// TIA Portal project "licznik-silownik" (V11)

(* hardware
DEVICE "S7-400 station_1"  S7400.Device
   slot 0: "UR1_0"  UR1  6ES7 400-1TA01-0AA0
   slot 2: "PLC_1"  CPU 416F-3 PN/DP  6ES7 416-3FR05-0AB0  V5.3
      slot 5: "PROFINET interface_1"  PN-IO
         slot 1: "Port_1"  Port
         slot 2: "Port_2"  Port
*)

// ===== PLC "PLC_1"  CPU 416F-3 PN/DP =====

VAR_GLOBAL   // PLC tag table "Default tag table"
   "Tag_1" AT %M0.0 : Bool;
   "Tag_2" AT %I0.0 : Bool;
   "Tag_3" AT %I0.1 : Bool;
   "Tag_4" AT %M1.0 : Bool;
   "Tag_5" AT %T1 : Timer;
   "Tag_6" AT %Q0.0 : Bool;
   "Tag_7" AT %M0.1 : Bool;
   "Tag_8" AT %M0.2 : Bool;
   "Tag_9" AT %I0.2 : Bool;
END_VAR

ORGANIZATION_BLOCK "Main"   // OB1, LAD
TITLE = "Main Program Sweep (Cycle)"
{ S7_Optimized_Access := 'FALSE' }
VERSION : 0.1
   VAR_TEMP
      OB1_EV_CLASS : Byte;   // Bits 0-3 = 1 (Coming event), Bits 4-7 = 1 (Event class 1)
      OB1_SCAN_1 : Byte;   // 1 (Cold restart scan 1 of OB 1), 3 (Scan 2-n of OB 1)
      OB1_PRIORITY : Byte;   // Priority of OB Execution
      OB1_OB_NUMBR : Byte;   // 1 (Organization block 1, OB1)
      OB1_RESERVED_1 : Byte;   // Reserved for system
      OB1_RESERVED_2 : Byte;   // Reserved for system
      OB1_PREV_CYCLE : Int;   // Cycle time of previous OB1 scan (milliseconds)
      OB1_MIN_CYCLE : Int;   // Minimum cycle time of OB1 (milliseconds)
      OB1_MAX_CYCLE : Int;   // Maximum cycle time of OB1 (milliseconds)
      OB1_DATE_TIME : Date_And_Time;   // Date and time OB1 started
   END_VAR
   VAR_TEMP   // added for the SCL form of the ladder/FBD networks
      _w1 : Bool;
      _s5time1 : S5Time;
   END_VAR
BEGIN

REGION Network 1
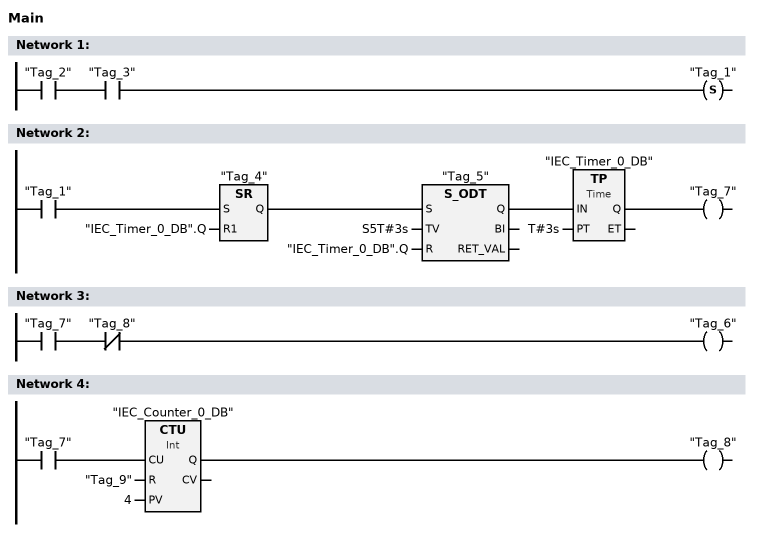
   RUNG wire#powerrail
      Contact( "Tag_2" )
      Contact( "Tag_3" )
      S_Coil( "Tag_1" )
   END_RUNG
   // the same network as SCL:
   IF "Tag_2" AND "Tag_3" THEN "Tag_1" := TRUE; END_IF;
END_REGION

REGION Network 2
   IF "Tag_1" THEN
       "Tag_4" := TRUE;   // SR flip-flop
   END_IF;
   IF "IEC_Timer_0_DB".Q THEN "Tag_4" := FALSE; END_IF;
   #_s5time1 := S_ODT(T_NO := "Tag_5", S := "Tag_4", TV := S5T#3s, R := "IEC_Timer_0_DB".Q, Q => #_w1);
   "IEC_Timer_0_DB".TP(IN := #_w1, PT := T#3s);
   "Tag_7" := "IEC_Timer_0_DB".Q;
END_REGION

REGION Network 3
   RUNG wire#powerrail
      Contact( "Tag_7" )
      I_Contact( "Tag_8" )
      Coil( "Tag_6" )
   END_RUNG
   // the same network as SCL:
   "Tag_6" := "Tag_7" AND NOT "Tag_8";
END_REGION

REGION Network 4
   "IEC_Counter_0_DB".CTU(CU := "Tag_7", R := "Tag_9", PV := 4);
   "Tag_8" := "IEC_Counter_0_DB".Q;
END_REGION
END_ORGANIZATION_BLOCK